FUNCTION_BLOCK FB_Error IMPLEMENTS I_State
VAR_INPUT
END_VAR
VAR_OUTPUT
END_VAR
VAR
	pAxis : POINTER TO FB_Axis;
END_VAR

{warning 'add method implementation '}
METHOD Disable : BOOL
END_METHOD

{warning 'add method implementation '}
METHOD Enable : BOOL
END_METHOD

METHOD FB_init : BOOL
VAR_INPUT
	bInitRetains : BOOL; // if TRUE, the retain variables are initialized (warm start / cold start)
	bInCopyCode : BOOL;  // if TRUE, the instance afterwards gets moved into the copy code (online change)
	pAxis : POINTER TO FB_Axis;
END_VAR
THIS^.pAxis := pAxis;
END_METHOD

{warning 'add method implementation '}
METHOD Reset : BOOL
END_METHOD

END_FUNCTION_BLOCK

(* stored: Version 1.1.0.1, ProductVersion 3.1.4024.3
   POU FB_Error: Id {580c34cd-9626-4b57-a2d4-b3ddeed16f6d}, SpecialFunc None
   Method Disable: Id {195830cd-6094-4844-b15d-b6cf2a074762}
   Method Enable: Id {12f833a1-36c3-40f8-b829-22cc6278629e}
   Method FB_init: Id {1f197484-3114-495c-9d8e-53e89fac3859}
   Method Reset: Id {3d993056-c150-474e-adcf-416ae6c805f4} *)
